ABB RobotStudio station: Practica3Avanzada_EstacionDePartida.rsstn

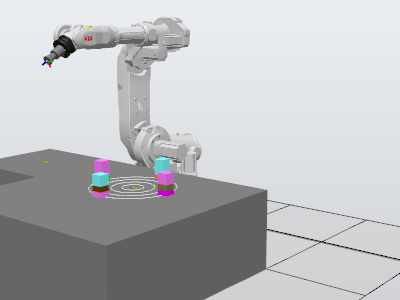
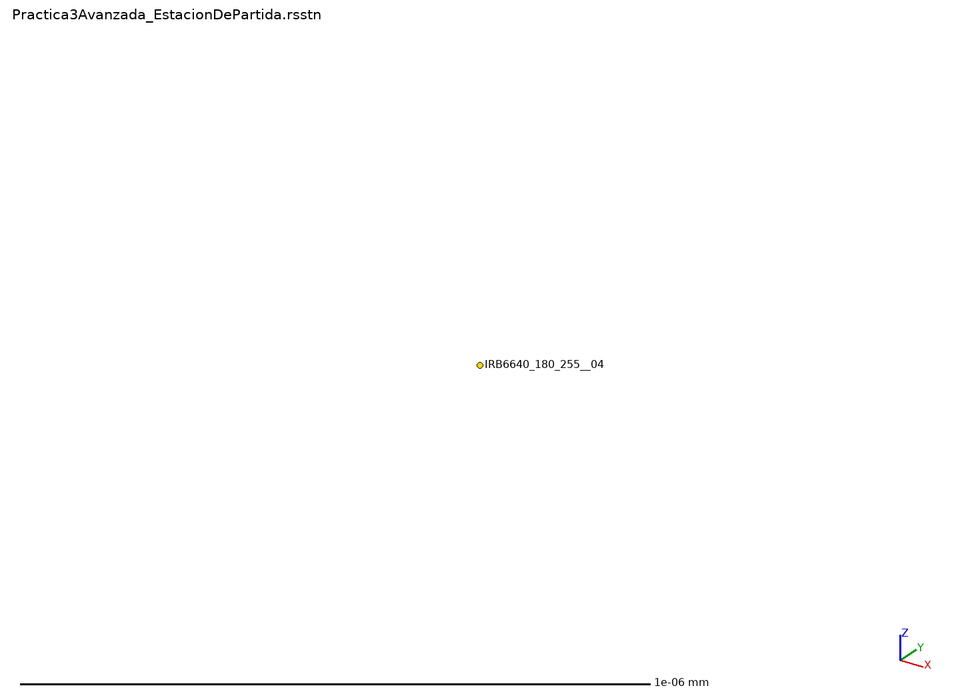
[picture v1: parts stored in the station drawn from their meshes, with robot base, taught points and paths (robot models come from the ABB library and are not in the file)]
Station Practica3Avanzada_EstacionDePartida (saved by RobotStudio 24.1.10713.1)
Controller Sistema6
  mechanical unit ROB_1: IRB6640_180_255__04, 6 joints, base frame (0, 0, 0) mm
Layout (positions relative to the parent item):
  - Ventosa [mechanism] at (1635.71, 0, 1955) mm, rotated rx 180 ry 60 rz 180 deg
      TCP Ventosa at (0, 0, 200) mm
      links: PiezaVentosa
  - IRB6640_180_255__04 [mechanism, from %ABB.RobotStudio.Models.IRB6640%\IRB6640_180_255_G_04.rslib] at (0, 0, 0) mm; joint values [0, 0, 0, 0, 0.5236, 0] (rad or m)
  - MesaTrabajoParte1 [part], size 1000 x 1000 x 750 mm
  - MesaTrabajoParte0 [part], size 1000 x 1000 x 750 mm
  - CI_VentosaVacuostato [smart component]
      signals: DI ActivaVentosa, DO Vacuostato
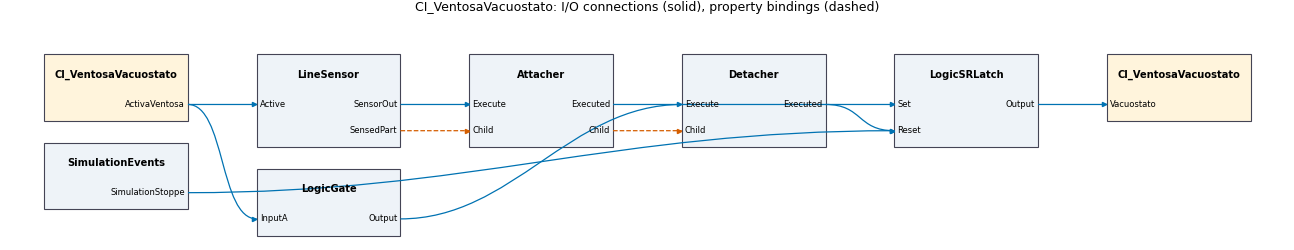
      connections:
        CI_VentosaVacuostato.ActivaVentosa -> LineSensor.Active
        LineSensor.SensorOut -> Attacher.Execute
        Attacher.Executed -> LogicSRLatch.Set
        LogicSRLatch.Output -> CI_VentosaVacuostato.Vacuostato
        Detacher.Executed -> LogicSRLatch.Reset
        SimulationEvents.SimulationStopped -> LogicSRLatch.Reset
        CI_VentosaVacuostato.ActivaVentosa -> LogicGate.InputA
        LogicGate.Output -> Detacher.Execute
        LineSensor.SensedPart => Attacher.Child
        Attacher.Child => Detacher.Child
    - LineSensor [smart component, from Components\LineSensor.rslib] at (1808.91, 0, 1855) mm, rotated rx 180 ry 60 rz 180 deg
        properties: Start=[0 0 -0.002]; End=[0 0 0.02]; Radius=0.002; SensedPart=Pieza1; SensedPoint=[1.69999987792969 0.6 0.95]; Length=0.022; Tag=(none)
      - _sensorPart_ [part], size 4 x 4 x 22 mm
    - SimulationEvents [smart component, from Components\SimulationEvents.rslib]
    - LogicSRLatch [smart component, from Components\LogicSRLatch.rslib]
    - Attacher [smart component, from Components\Attacher.rslib]
        properties: Parent=Ventosa; Flange=0; Child=Pieza1; Mount=false; Offset=[0 0 0]; Orientation=[0 0 0]
    - Detacher [smart component, from Components\Detacher.rslib]
        properties: Child=Pieza1; KeepPosition=true
    - LogicGate [smart component, from Components\LogicGate.rslib]
        properties: Operator=NOT; Delay=0.1
  - MesaTrabajoParte2 [part] at (0, 1000, 0) mm, size 1000 x 1000 x 750 mm
  - MesaTrabajoParte3 [part] at (1000, 0, 0) mm, size 1000 x 1000 x 750 mm
  - MesaTrabajoParte4 [part] at (1000, 1000, 0) mm, size 1000 x 1000 x 750 mm
  - Pieza1 [part] at (200, 1100, 150) mm, size 100 x 100 x 50 mm
  - Pieza2 [part] at (-200, 1500, 100) mm, size 100 x 100 x 50 mm
  - Pieza3 [part] at (200, 1900, 50) mm, size 100 x 100 x 50 mm
  - Pieza4 [part] at (600, 1500, 0) mm, size 100 x 100 x 50 mm
  - Pieza5 [part] at (200, 1100, -100) mm, size 100 x 100 x 50 mm
  - CircunferenciaR200 [part], size 400 x 400 x 0 mm
  - CircunferenciaR100 [part], size 200 x 198.9 x 0 mm
  - CircunferenciaR300 [part], size 599 x 599.5 x 0 mm
  - CircunferenciaR400 [part], size 799 x 799.5 x 0 mm
  - Pieza6 [part] at (-200, 1500, -150) mm, size 100 x 100 x 50 mm
  - Pieza7 [part] at (200, 1900, -200) mm, size 100 x 100 x 50 mm
  - Pieza8 [part] at (600, 1500, -250) mm, size 100 x 100 x 50 mm
  - Pieza9 [part] at (200, 1100, -350) mm, size 100 x 100 x 50 mm
  - Pieza10 [part] at (-200, 1500, -400) mm, size 100 x 100 x 50 mm
  - Pieza10_2 [part] at (200, 1900, -400) mm, size 100 x 100 x 50 mm
  - Pieza10_5 [part] at (600, 1500, -400) mm, size 100 x 100 x 50 mm
  - Pieza10_6 [part] at (200, 1100, -450) mm, size 100 x 100 x 50 mm
  - Pieza10_7 [part] at (-200, 1500, -450) mm, size 100 x 100 x 50 mm
  - Pieza10_8 [part] at (200, 1900, -450) mm, size 100 x 100 x 50 mm
  - Pieza10_9 [part] at (600, 1500, -450) mm, size 100 x 100 x 50 mm
Attachment: Ventosa is attached to IRB6640_180_255__04 / Link6
Attachment: LineSensor is attached to Ventosa / PiezaVentosa
Station logic (signal -> signal, property => property):
  CI_VentosaVacuostato.Vacuostato -> Sistema6.ED_PiezaCogida
  Sistema6.SD_ActivaVentosa -> CI_VentosaVacuostato.ActivaVentosa
Targets, tools, work objects and paths stored in the station, written as RAPID:
! task T_ROB1
MODULE CalibData
  PERS tooldata Ventosa:=[TRUE,[[0,0,200],[1,0,0,0]],[1,[0,0,125],[1,0,0,0],0.002,0.002,0.0013]];
ENDMODULE

! task T_ROB1
MODULE Module1
  CONST robtarget pBaseOrigen:=[[1500,-500,750],[0,0,1,0],[0,0,0,0],[9E+09,9E+09,9E+09,9E+09,9E+09,9E+09]];
  CONST robtarget pCentroDestino:=[[1700,1000,750],[0,0,1,0],[0,0,0,0],[9E+09,9E+09,9E+09,9E+09,9E+09,9E+09]];
  CONST robtarget pReposo:=[[1808.910161514,0,1855],[0.5,0,0.866025404,0],[0,0,0,0],[9E+09,9E+09,9E+09,9E+09,9E+09,9E+09]];
ENDMODULE

